TYPE TcaPushButtonRef :
STRUCT
	Button AT%I* : BOOL;
	Light AT%Q* : BOOL;	
END_STRUCT
END_TYPE

(* stored: Version 1.1.0.1
   DUT TcaPushButtonRef: Id {f5896e44-9448-4821-87d6-90bc34c4bdca} *)
